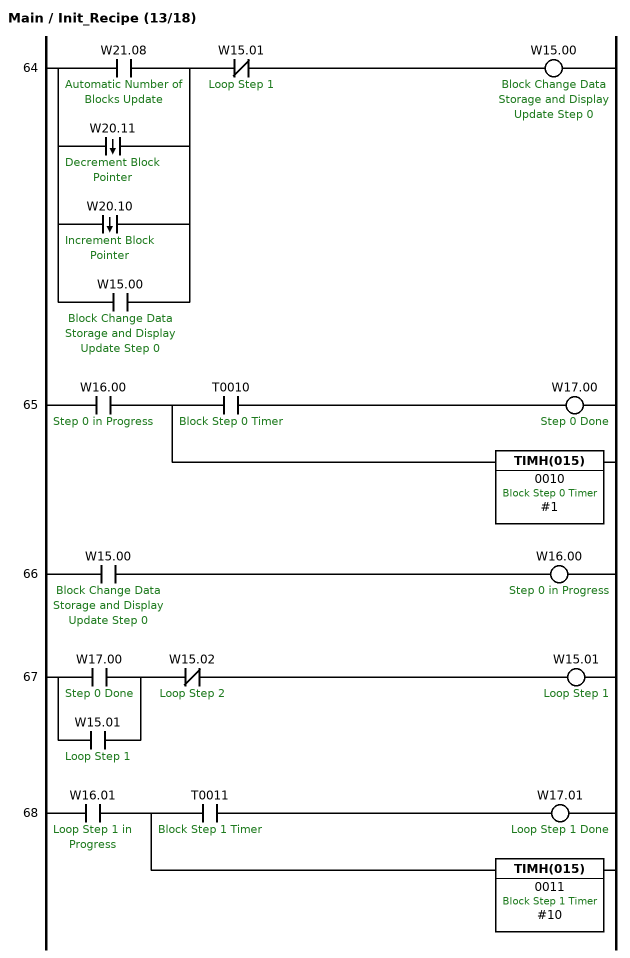
; [picture p72: Main / Init_Recipe, rungs 64-68]
; rung 64
LD W21.08  ; Automatic Number of Blocks Update
%OR W20.11  ; Decrement Block Pointer
%OR W20.10  ; Increment Block Pointer
OR W15.00  ; Block Change Data Storage and Display Update Step 0
ANDNOT W15.01  ; Loop Step 1
OUT W15.00  ; Block Change Data Storage and Display Update Step 0
; rung 65
LD W16.00  ; Step 0 in Progress
OUT TR0
AND T0010  ; Block Step 0 Timer
OUT W17.00  ; Step 0 Done
LD TR0
TIMH(015) 0010 #1  ; Block Step 0 Timer
; rung 66
LD W15.00  ; Block Change Data Storage and Display Update Step 0
OUT W16.00  ; Step 0 in Progress
; rung 67
LD W17.00  ; Step 0 Done
OR W15.01  ; Loop Step 1
ANDNOT W15.02  ; Loop Step 2
OUT W15.01  ; Loop Step 1
; rung 68
LD W16.01  ; Loop Step 1 in Progress
OUT TR0
AND T0011  ; Block Step 1 Timer
OUT W17.01  ; Loop Step 1 Done
LD TR0
TIMH(015) 0011 #10  ; Block Step 1 Timer

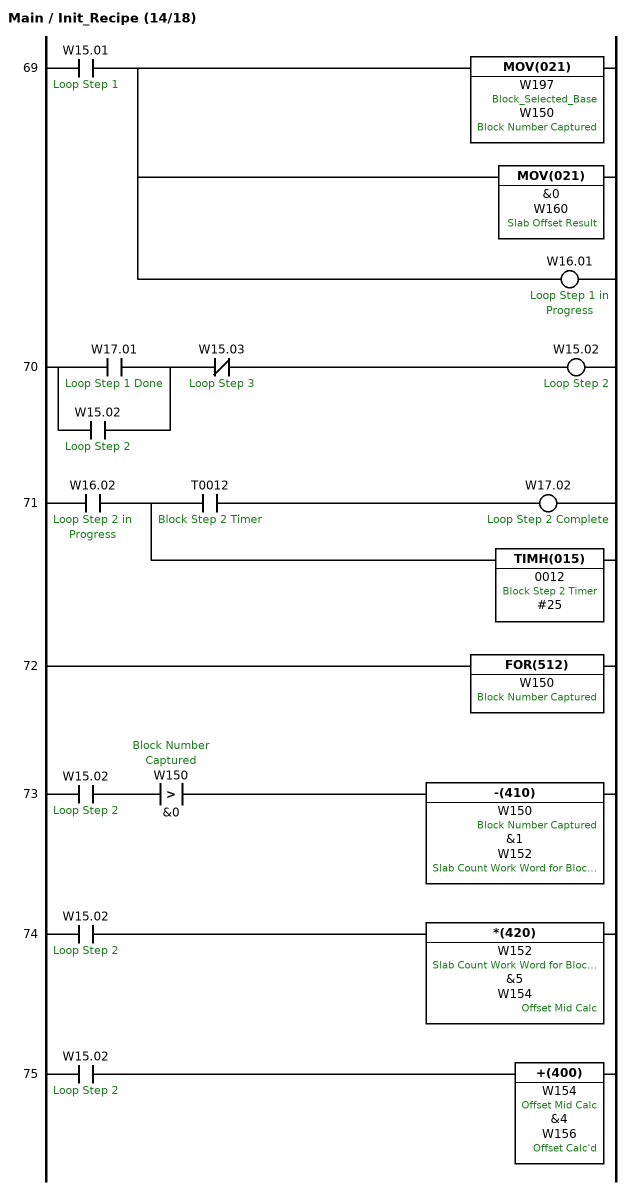
; rung 69
LD W15.01  ; Loop Step 1
MOV(021) W197 W150  ; Block_Selected_Base, Block Number Captured
MOV(021) &0 W160  ; Slab Offset Result
OUT W16.01  ; Loop Step 1 in Progress
; rung 70
LD W17.01  ; Loop Step 1 Done
OR W15.02  ; Loop Step 2
ANDNOT W15.03  ; Loop Step 3
OUT W15.02  ; Loop Step 2
; rung 71
LD W16.02  ; Loop Step 2 in Progress
OUT TR0
AND T0012  ; Block Step 2 Timer
OUT W17.02  ; Loop Step 2 Complete
LD TR0
TIMH(015) 0012 #25  ; Block Step 2 Timer
; rung 72
FOR(512) W150  ; Block Number Captured
; rung 73
LD W15.02  ; Loop Step 2
AND>(320) W150 &0  ; Block Number Captured
-(410) W150 &1 W152  ; Block Number Captured, Slab Count Work Word for Block Pointer
; rung 74
LD W15.02  ; Loop Step 2
*(420) W152 &5 W154  ; Slab Count Work Word for Block Pointer, Offset Mid Calc
; rung 75
LD W15.02  ; Loop Step 2
+(400) W154 &4 W156  ; Offset Mid Calc, Offset Calc'd

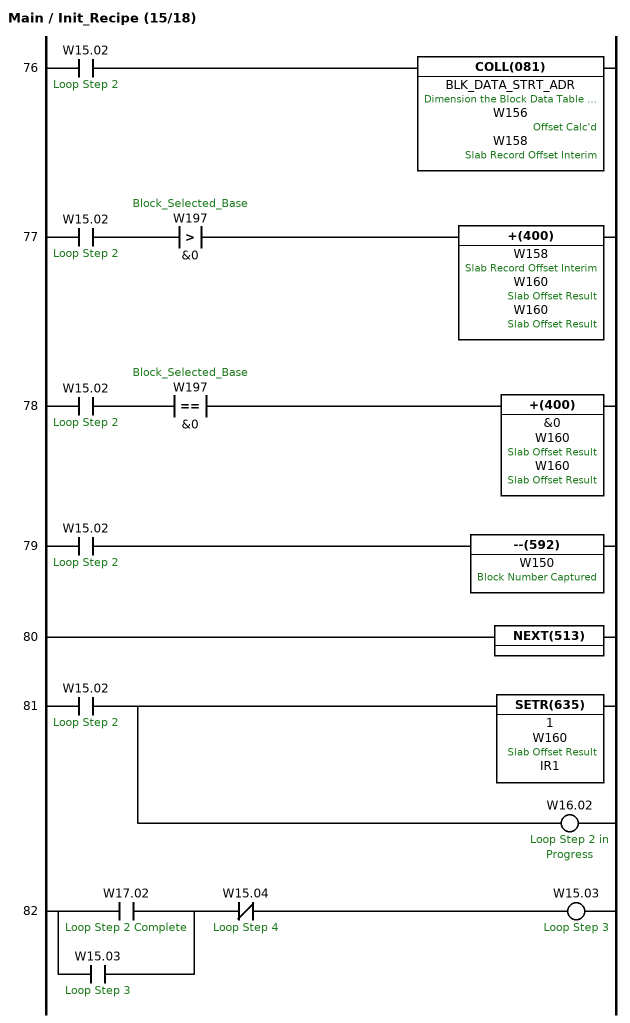
; rung 76
LD W15.02  ; Loop Step 2
COLL(081) BLK_DATA_STRT_ADR W156 W158  ; Dimension the Block Data Table - Start Address, Offset Calc'd, Slab Record Offset Interim
; rung 77
LD W15.02  ; Loop Step 2
AND>(320) W197 &0  ; Block_Selected_Base
+(400) W158 W160 W160  ; Slab Record Offset Interim, Slab Offset Result
; rung 78
LD W15.02  ; Loop Step 2
AND=(300) W197 &0  ; Block_Selected_Base
+(400) &0 W160 W160  ; Slab Offset Result
; rung 79
LD W15.02  ; Loop Step 2
--(592) W150  ; Block Number Captured
; rung 80
NEXT(513)
; rung 81
LD W15.02  ; Loop Step 2
SETR(635) 1 W160 IR1  ; Slab Offset Result
OUT W16.02  ; Loop Step 2 in Progress
; rung 82
LD W17.02  ; Loop Step 2 Complete
OR W15.03  ; Loop Step 3
ANDNOT W15.04  ; Loop Step 4
OUT W15.03  ; Loop Step 3

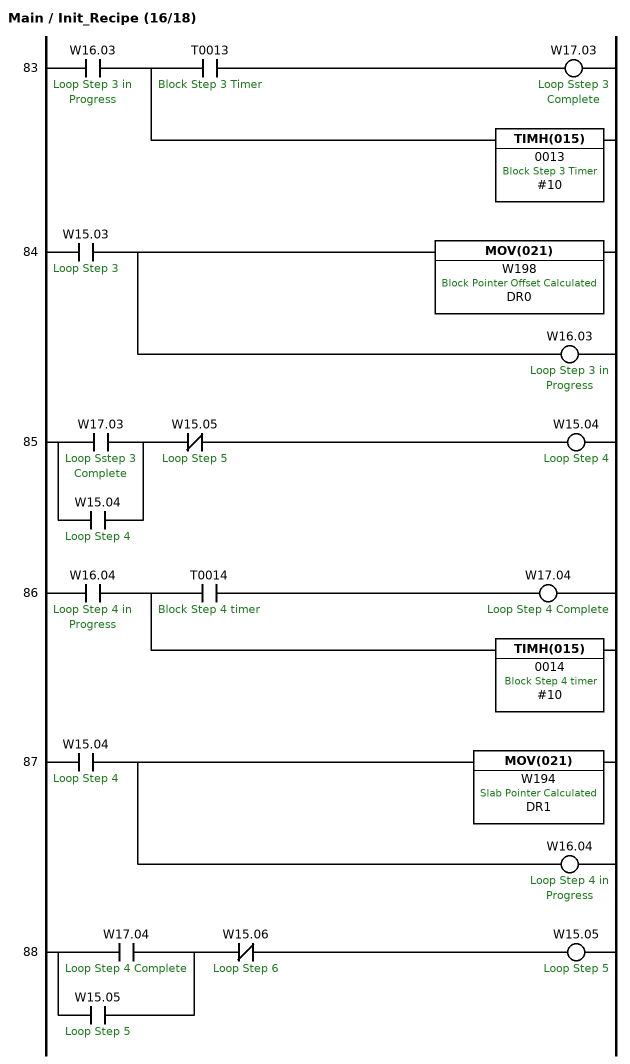
; rung 83
LD W16.03  ; Loop Step 3 in Progress
OUT TR0
AND T0013  ; Block Step 3 Timer
OUT W17.03  ; Loop Sstep 3 Complete
LD TR0
TIMH(015) 0013 #10  ; Block Step 3 Timer
; rung 84
LD W15.03  ; Loop Step 3
MOV(021) W198 DR0  ; Block Pointer Offset Calculated
OUT W16.03  ; Loop Step 3 in Progress
; rung 85
LD W17.03  ; Loop Sstep 3 Complete
OR W15.04  ; Loop Step 4
ANDNOT W15.05  ; Loop Step 5
OUT W15.04  ; Loop Step 4
; rung 86
LD W16.04  ; Loop Step 4 in Progress
OUT TR0
AND T0014  ; Block Step 4 timer
OUT W17.04  ; Loop Step 4 Complete
LD TR0
TIMH(015) 0014 #10  ; Block Step 4 timer
; rung 87
LD W15.04  ; Loop Step 4
MOV(021) W194 DR1  ; Slab Pointer Calculated
OUT W16.04  ; Loop Step 4 in Progress
; rung 88
LD W17.04  ; Loop Step 4 Complete
OR W15.05  ; Loop Step 5
ANDNOT W15.06  ; Loop Step 6
OUT W15.05  ; Loop Step 5

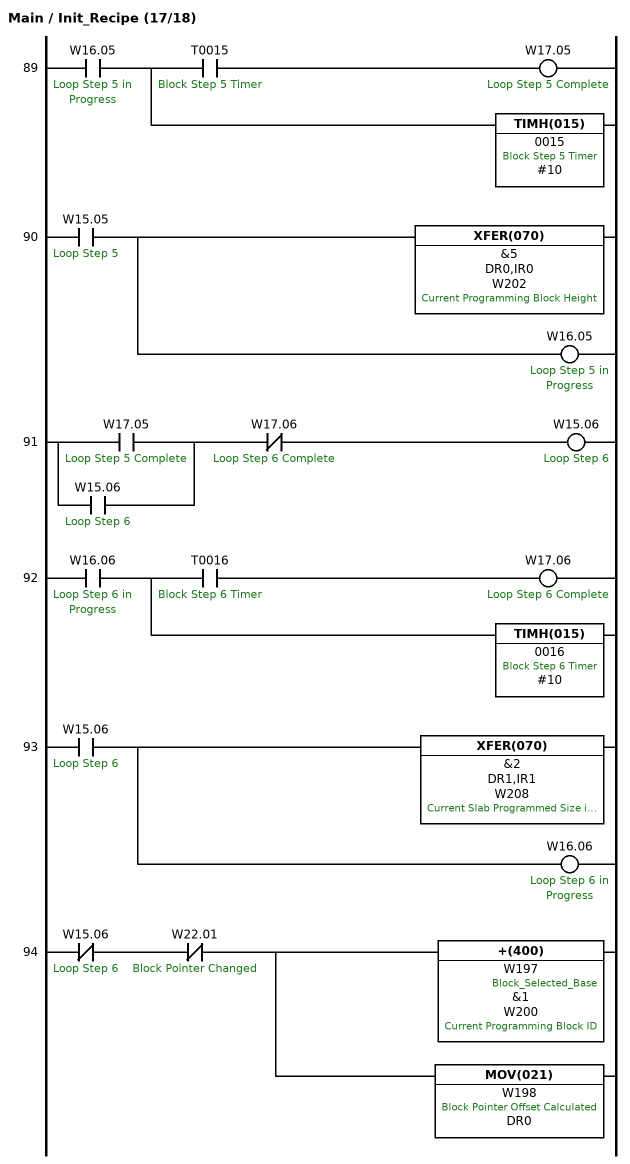
; rung 89
LD W16.05  ; Loop Step 5 in Progress
OUT TR0
AND T0015  ; Block Step 5 Timer
OUT W17.05  ; Loop Step 5 Complete
LD TR0
TIMH(015) 0015 #10  ; Block Step 5 Timer
; rung 90
LD W15.05  ; Loop Step 5
XFER(070) &5 DR0,IR0 W202  ; Current Programming Block Height
OUT W16.05  ; Loop Step 5 in Progress
; rung 91
LD W17.05  ; Loop Step 5 Complete
OR W15.06  ; Loop Step 6
ANDNOT W17.06  ; Loop Step 6 Complete
OUT W15.06  ; Loop Step 6
; rung 92
LD W16.06  ; Loop Step 6 in Progress
OUT TR0
AND T0016  ; Block Step 6 Timer
OUT W17.06  ; Loop Step 6 Complete
LD TR0
TIMH(015) 0016 #10  ; Block Step 6 Timer
; rung 93
LD W15.06  ; Loop Step 6
XFER(070) &2 DR1,IR1 W208  ; Current Slab Programmed Size in inches
OUT W16.06  ; Loop Step 6 in Progress
; rung 94
LDNOT W15.06  ; Loop Step 6
ANDNOT W22.01  ; Block Pointer Changed
+(400) W197 &1 W200  ; Block_Selected_Base, Current Programming Block ID
MOV(021) W198 DR0  ; Block Pointer Offset Calculated

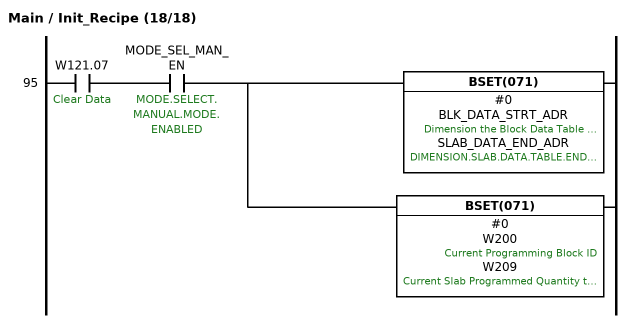
; rung 95
LD W121.07  ; Clear Data
AND MODE_SEL_MAN_EN  ; MODE.SELECT.MANUAL.MODE.ENABLED
BSET(071) #0 BLK_DATA_STRT_ADR SLAB_DATA_END_ADR  ; Dimension the Block Data Table - Start Address, DIMENSION.SLAB.DATA.TABLE.END.ADDRESS
BSET(071) #0 W200 W209  ; Current Programming Block ID, Current Slab Programmed Quantity to cut

### Section Init_Message_Display

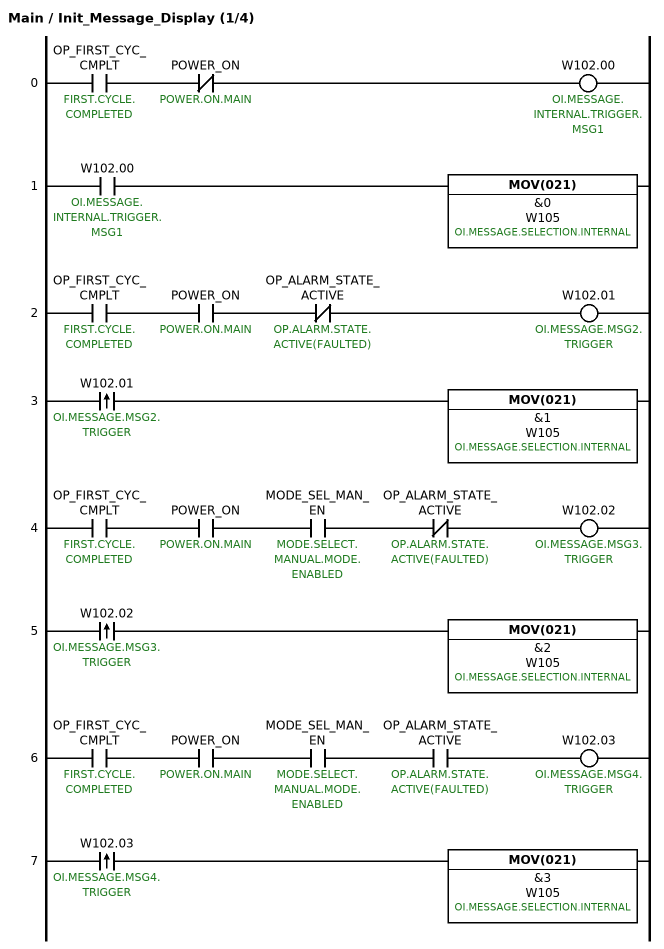
; rung 0
LD OP_FIRST_CYC_CMPLT  ; FIRST.CYCLE.COMPLETED
ANDNOT POWER_ON  ; POWER.ON.MAIN
OUT W102.00  ; OI.MESSAGE.INTERNAL.TRIGGER.MSG1
; rung 1
LD W102.00  ; OI.MESSAGE.INTERNAL.TRIGGER.MSG1
MOV(021) &0 W105  ; OI.MESSAGE.SELECTION.INTERNAL
; rung 2
LD OP_FIRST_CYC_CMPLT  ; FIRST.CYCLE.COMPLETED
AND POWER_ON  ; POWER.ON.MAIN
ANDNOT OP_ALARM_STATE_ACTIVE  ; OP.ALARM.STATE.ACTIVE(FAULTED)
OUT W102.01  ; OI.MESSAGE.MSG2.TRIGGER
; rung 3
@LD W102.01  ; OI.MESSAGE.MSG2.TRIGGER
MOV(021) &1 W105  ; OI.MESSAGE.SELECTION.INTERNAL
; rung 4
LD OP_FIRST_CYC_CMPLT  ; FIRST.CYCLE.COMPLETED
AND POWER_ON  ; POWER.ON.MAIN
AND MODE_SEL_MAN_EN  ; MODE.SELECT.MANUAL.MODE.ENABLED
ANDNOT OP_ALARM_STATE_ACTIVE  ; OP.ALARM.STATE.ACTIVE(FAULTED)
OUT W102.02  ; OI.MESSAGE.MSG3.TRIGGER
; rung 5
@LD W102.02  ; OI.MESSAGE.MSG3.TRIGGER
MOV(021) &2 W105  ; OI.MESSAGE.SELECTION.INTERNAL
; rung 6
LD OP_FIRST_CYC_CMPLT  ; FIRST.CYCLE.COMPLETED
AND POWER_ON  ; POWER.ON.MAIN
AND MODE_SEL_MAN_EN  ; MODE.SELECT.MANUAL.MODE.ENABLED
AND OP_ALARM_STATE_ACTIVE  ; OP.ALARM.STATE.ACTIVE(FAULTED)
OUT W102.03  ; OI.MESSAGE.MSG4.TRIGGER
; rung 7
@LD W102.03  ; OI.MESSAGE.MSG4.TRIGGER
MOV(021) &3 W105  ; OI.MESSAGE.SELECTION.INTERNAL

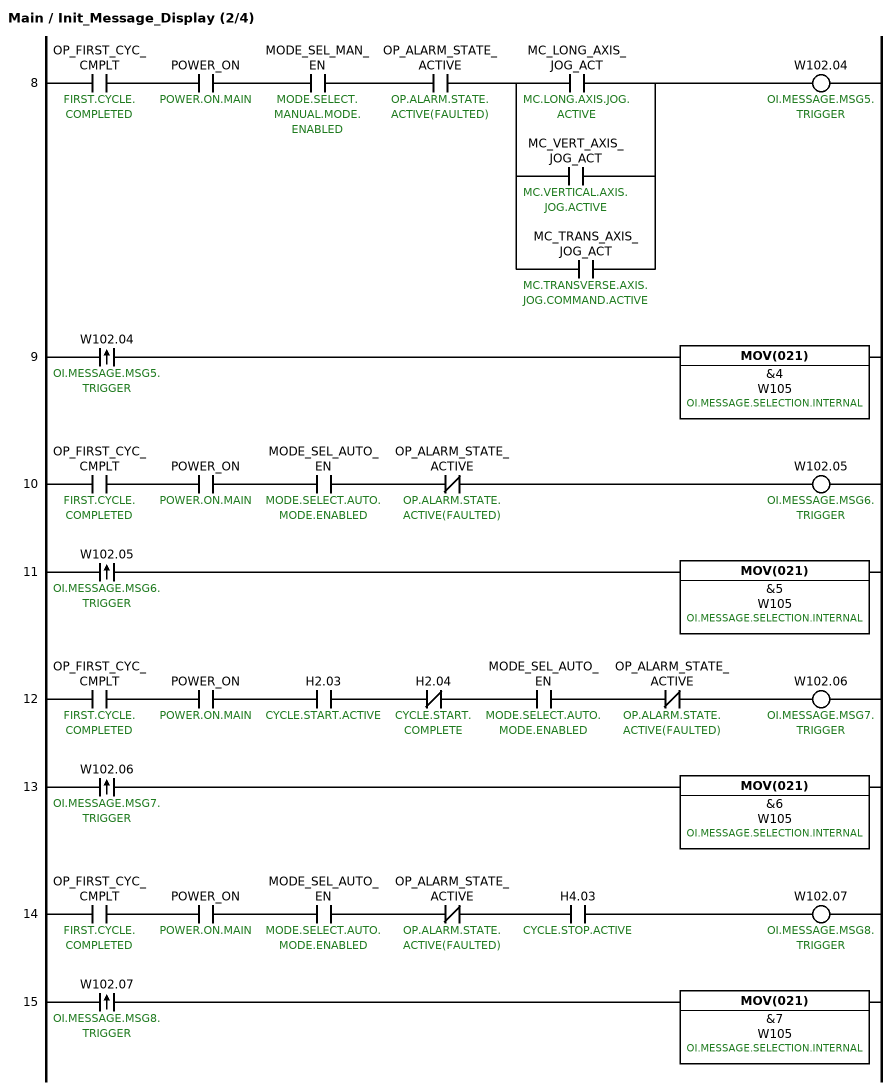
; rung 8
LD OP_FIRST_CYC_CMPLT  ; FIRST.CYCLE.COMPLETED
AND POWER_ON  ; POWER.ON.MAIN
AND MODE_SEL_MAN_EN  ; MODE.SELECT.MANUAL.MODE.ENABLED
AND OP_ALARM_STATE_ACTIVE  ; OP.ALARM.STATE.ACTIVE(FAULTED)
LD MC_LONG_AXIS_JOG_ACT  ; MC.LONG.AXIS.JOG.ACTIVE
OR MC_VERT_AXIS_JOG_ACT  ; MC.VERTICAL.AXIS.JOG.ACTIVE
OR MC_TRANS_AXIS_JOG_ACT  ; MC.TRANSVERSE.AXIS.JOG.COMMAND.ACTIVE
ANDLD
OUT W102.04  ; OI.MESSAGE.MSG5.TRIGGER
; rung 9
@LD W102.04  ; OI.MESSAGE.MSG5.TRIGGER
MOV(021) &4 W105  ; OI.MESSAGE.SELECTION.INTERNAL
; rung 10
LD OP_FIRST_CYC_CMPLT  ; FIRST.CYCLE.COMPLETED
AND POWER_ON  ; POWER.ON.MAIN
AND MODE_SEL_AUTO_EN  ; MODE.SELECT.AUTO.MODE.ENABLED
ANDNOT OP_ALARM_STATE_ACTIVE  ; OP.ALARM.STATE.ACTIVE(FAULTED)
OUT W102.05  ; OI.MESSAGE.MSG6.TRIGGER
; rung 11
@LD W102.05  ; OI.MESSAGE.MSG6.TRIGGER
MOV(021) &5 W105  ; OI.MESSAGE.SELECTION.INTERNAL
; rung 12
LD OP_FIRST_CYC_CMPLT  ; FIRST.CYCLE.COMPLETED
AND POWER_ON  ; POWER.ON.MAIN
AND H2.03  ; CYCLE.START.ACTIVE
ANDNOT H2.04  ; CYCLE.START.COMPLETE
AND MODE_SEL_AUTO_EN  ; MODE.SELECT.AUTO.MODE.ENABLED
ANDNOT OP_ALARM_STATE_ACTIVE  ; OP.ALARM.STATE.ACTIVE(FAULTED)
OUT W102.06  ; OI.MESSAGE.MSG7.TRIGGER
; rung 13
@LD W102.06  ; OI.MESSAGE.MSG7.TRIGGER
MOV(021) &6 W105  ; OI.MESSAGE.SELECTION.INTERNAL
; rung 14
LD OP_FIRST_CYC_CMPLT  ; FIRST.CYCLE.COMPLETED
AND POWER_ON  ; POWER.ON.MAIN
AND MODE_SEL_AUTO_EN  ; MODE.SELECT.AUTO.MODE.ENABLED
ANDNOT OP_ALARM_STATE_ACTIVE  ; OP.ALARM.STATE.ACTIVE(FAULTED)
AND H4.03  ; CYCLE.STOP.ACTIVE
OUT W102.07  ; OI.MESSAGE.MSG8.TRIGGER
; rung 15
@LD W102.07  ; OI.MESSAGE.MSG8.TRIGGER
MOV(021) &7 W105  ; OI.MESSAGE.SELECTION.INTERNAL

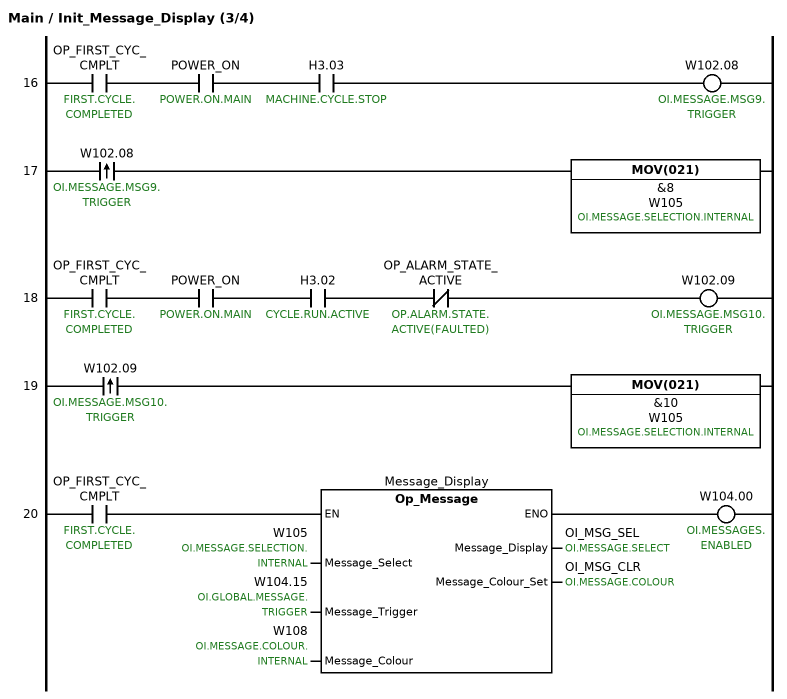
; rung 16
LD OP_FIRST_CYC_CMPLT  ; FIRST.CYCLE.COMPLETED
AND POWER_ON  ; POWER.ON.MAIN
AND H3.03  ; MACHINE.CYCLE.STOP
OUT W102.08  ; OI.MESSAGE.MSG9.TRIGGER
; rung 17
@LD W102.08  ; OI.MESSAGE.MSG9.TRIGGER
MOV(021) &8 W105  ; OI.MESSAGE.SELECTION.INTERNAL
; rung 18
LD OP_FIRST_CYC_CMPLT  ; FIRST.CYCLE.COMPLETED
AND POWER_ON  ; POWER.ON.MAIN
AND H3.02  ; CYCLE.RUN.ACTIVE
ANDNOT OP_ALARM_STATE_ACTIVE  ; OP.ALARM.STATE.ACTIVE(FAULTED)
OUT W102.09  ; OI.MESSAGE.MSG10.TRIGGER
; rung 19
@LD W102.09  ; OI.MESSAGE.MSG10.TRIGGER
MOV(021) &10 W105  ; OI.MESSAGE.SELECTION.INTERNAL
; rung 20
LD OP_FIRST_CYC_CMPLT  ; FIRST.CYCLE.COMPLETED
CALL Message_Display : Op_Message (Message_Select := W105, Message_Trigger := W104.15, Message_Colour := W108, Message_Display => OI_MSG_SEL, Message_Colour_Set => OI_MSG_CLR)  ; OI.MESSAGE.SELECTION.INTERNAL, OI.GLOBAL.MESSAGE.TRIGGER, OI.MESSAGE.COLOUR.INTERNAL, OI.MESSAGE.SELECT, OI.MESSAGE.COLOUR
OUT W104.00  ; OI.MESSAGES.ENABLED

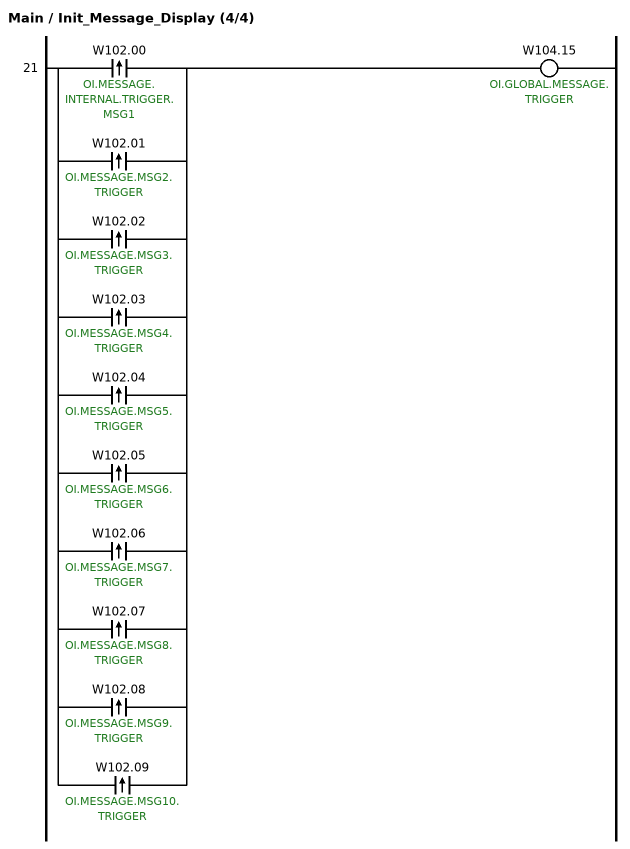
; rung 21
@LD W102.00  ; OI.MESSAGE.INTERNAL.TRIGGER.MSG1
@OR W102.01  ; OI.MESSAGE.MSG2.TRIGGER
@OR W102.02  ; OI.MESSAGE.MSG3.TRIGGER
@OR W102.03  ; OI.MESSAGE.MSG4.TRIGGER
@OR W102.04  ; OI.MESSAGE.MSG5.TRIGGER
@OR W102.05  ; OI.MESSAGE.MSG6.TRIGGER
@OR W102.06  ; OI.MESSAGE.MSG7.TRIGGER
@OR W102.07  ; OI.MESSAGE.MSG8.TRIGGER
@OR W102.08  ; OI.MESSAGE.MSG9.TRIGGER
@OR W102.09  ; OI.MESSAGE.MSG10.TRIGGER
OUT W104.15  ; OI.GLOBAL.MESSAGE.TRIGGER

### Section Init_Alarm_Display

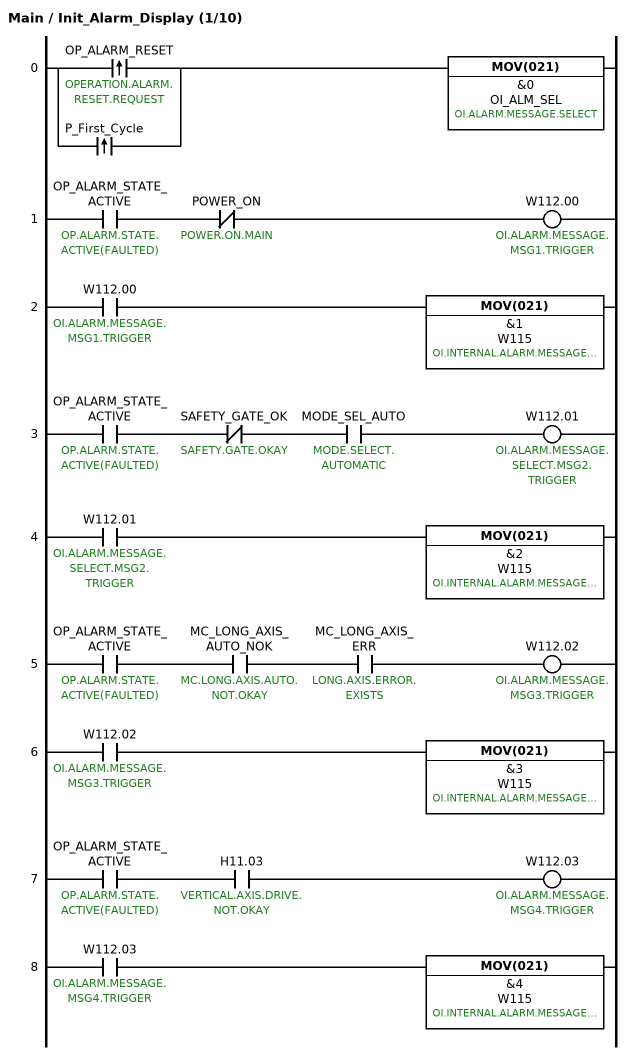
; rung 0
@LD OP_ALARM_RESET  ; OPERATION.ALARM.RESET.REQUEST
@OR P_First_Cycle
MOV(021) &0 OI_ALM_SEL  ; OI.ALARM.MESSAGE.SELECT
; rung 1
LD OP_ALARM_STATE_ACTIVE  ; OP.ALARM.STATE.ACTIVE(FAULTED)
ANDNOT POWER_ON  ; POWER.ON.MAIN
OUT W112.00  ; OI.ALARM.MESSAGE.MSG1.TRIGGER
; rung 2
LD W112.00  ; OI.ALARM.MESSAGE.MSG1.TRIGGER
MOV(021) &1 W115  ; OI.INTERNAL.ALARM.MESSAGE.SELECTION
; rung 3
LD OP_ALARM_STATE_ACTIVE  ; OP.ALARM.STATE.ACTIVE(FAULTED)
ANDNOT SAFETY_GATE_OK  ; SAFETY.GATE.OKAY
AND MODE_SEL_AUTO  ; MODE.SELECT.AUTOMATIC
OUT W112.01  ; OI.ALARM.MESSAGE.SELECT.MSG2.TRIGGER
; rung 4
LD W112.01  ; OI.ALARM.MESSAGE.SELECT.MSG2.TRIGGER
MOV(021) &2 W115  ; OI.INTERNAL.ALARM.MESSAGE.SELECTION
; rung 5
LD OP_ALARM_STATE_ACTIVE  ; OP.ALARM.STATE.ACTIVE(FAULTED)
AND MC_LONG_AXIS_AUTO_NOK  ; MC.LONG.AXIS.AUTO.NOT.OKAY
AND MC_LONG_AXIS_ERR  ; LONG.AXIS.ERROR.EXISTS
OUT W112.02  ; OI.ALARM.MESSAGE.MSG3.TRIGGER
; rung 6
LD W112.02  ; OI.ALARM.MESSAGE.MSG3.TRIGGER
MOV(021) &3 W115  ; OI.INTERNAL.ALARM.MESSAGE.SELECTION
; rung 7
LD OP_ALARM_STATE_ACTIVE  ; OP.ALARM.STATE.ACTIVE(FAULTED)
AND H11.03  ; VERTICAL.AXIS.DRIVE.NOT.OKAY
OUT W112.03  ; OI.ALARM.MESSAGE.MSG4.TRIGGER
; rung 8
LD W112.03  ; OI.ALARM.MESSAGE.MSG4.TRIGGER
MOV(021) &4 W115  ; OI.INTERNAL.ALARM.MESSAGE.SELECTION

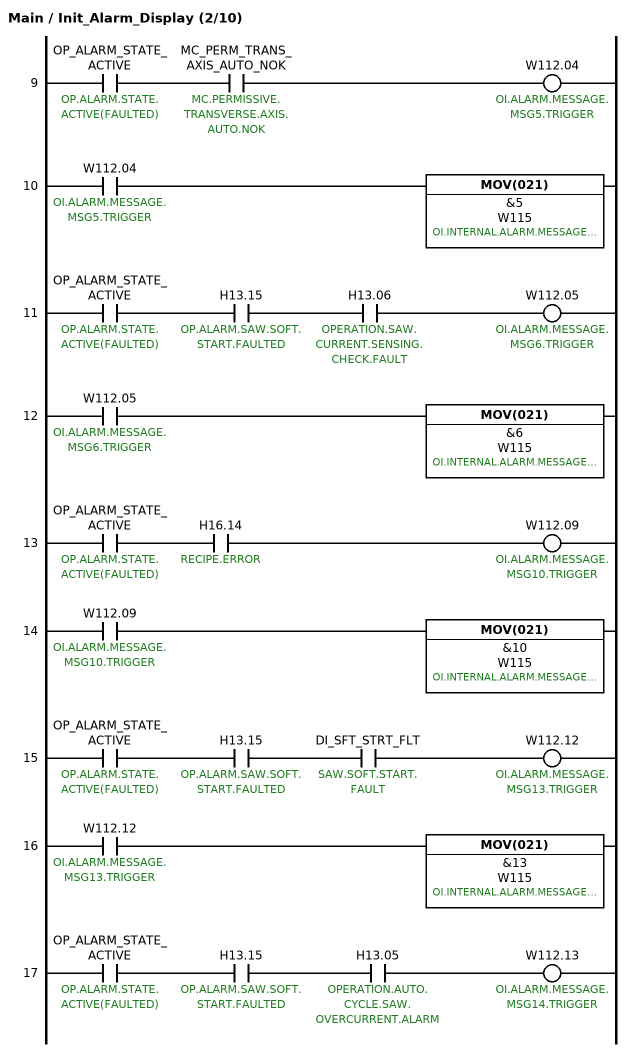
; rung 9
LD OP_ALARM_STATE_ACTIVE  ; OP.ALARM.STATE.ACTIVE(FAULTED)
AND MC_PERM_TRANS_AXIS_AUTO_NOK  ; MC.PERMISSIVE.TRANSVERSE.AXIS.AUTO.NOK
OUT W112.04  ; OI.ALARM.MESSAGE.MSG5.TRIGGER
; rung 10
LD W112.04  ; OI.ALARM.MESSAGE.MSG5.TRIGGER
MOV(021) &5 W115  ; OI.INTERNAL.ALARM.MESSAGE.SELECTION
; rung 11
LD OP_ALARM_STATE_ACTIVE  ; OP.ALARM.STATE.ACTIVE(FAULTED)
AND H13.15  ; OP.ALARM.SAW.SOFT.START.FAULTED
AND H13.06  ; OPERATION.SAW.CURRENT.SENSING.CHECK.FAULT
OUT W112.05  ; OI.ALARM.MESSAGE.MSG6.TRIGGER
; rung 12
LD W112.05  ; OI.ALARM.MESSAGE.MSG6.TRIGGER
MOV(021) &6 W115  ; OI.INTERNAL.ALARM.MESSAGE.SELECTION
; rung 13
LD OP_ALARM_STATE_ACTIVE  ; OP.ALARM.STATE.ACTIVE(FAULTED)
AND H16.14  ; RECIPE.ERROR
OUT W112.09  ; OI.ALARM.MESSAGE.MSG10.TRIGGER
; rung 14
LD W112.09  ; OI.ALARM.MESSAGE.MSG10.TRIGGER
MOV(021) &10 W115  ; OI.INTERNAL.ALARM.MESSAGE.SELECTION
; rung 15
LD OP_ALARM_STATE_ACTIVE  ; OP.ALARM.STATE.ACTIVE(FAULTED)
AND H13.15  ; OP.ALARM.SAW.SOFT.START.FAULTED
AND DI_SFT_STRT_FLT  ; SAW.SOFT.START.FAULT
OUT W112.12  ; OI.ALARM.MESSAGE.MSG13.TRIGGER
; rung 16
LD W112.12  ; OI.ALARM.MESSAGE.MSG13.TRIGGER
MOV(021) &13 W115  ; OI.INTERNAL.ALARM.MESSAGE.SELECTION
; rung 17
LD OP_ALARM_STATE_ACTIVE  ; OP.ALARM.STATE.ACTIVE(FAULTED)
AND H13.15  ; OP.ALARM.SAW.SOFT.START.FAULTED
AND H13.05  ; OPERATION.AUTO.CYCLE.SAW.OVERCURRENT.ALARM
OUT W112.13  ; OI.ALARM.MESSAGE.MSG14.TRIGGER

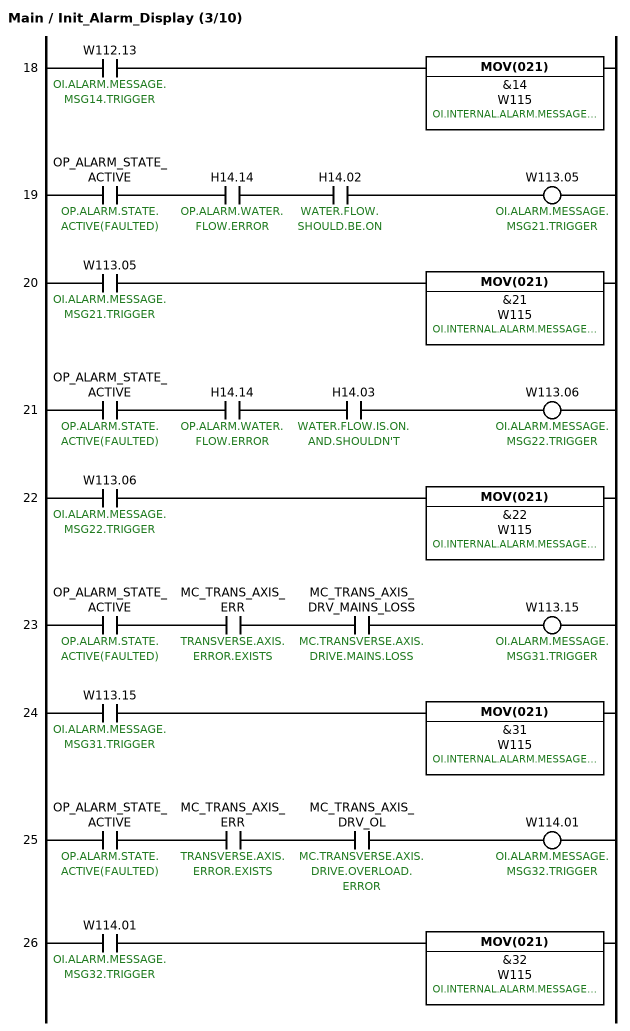
; rung 18
LD W112.13  ; OI.ALARM.MESSAGE.MSG14.TRIGGER
MOV(021) &14 W115  ; OI.INTERNAL.ALARM.MESSAGE.SELECTION
; rung 19
LD OP_ALARM_STATE_ACTIVE  ; OP.ALARM.STATE.ACTIVE(FAULTED)
AND H14.14  ; OP.ALARM.WATER.FLOW.ERROR
AND H14.02  ; WATER.FLOW.SHOULD.BE.ON
OUT W113.05  ; OI.ALARM.MESSAGE.MSG21.TRIGGER
; rung 20
LD W113.05  ; OI.ALARM.MESSAGE.MSG21.TRIGGER
MOV(021) &21 W115  ; OI.INTERNAL.ALARM.MESSAGE.SELECTION
; rung 21
LD OP_ALARM_STATE_ACTIVE  ; OP.ALARM.STATE.ACTIVE(FAULTED)
AND H14.14  ; OP.ALARM.WATER.FLOW.ERROR
AND H14.03  ; WATER.FLOW.IS.ON.AND.SHOULDN'T
OUT W113.06  ; OI.ALARM.MESSAGE.MSG22.TRIGGER
; rung 22
LD W113.06  ; OI.ALARM.MESSAGE.MSG22.TRIGGER
MOV(021) &22 W115  ; OI.INTERNAL.ALARM.MESSAGE.SELECTION
; rung 23
LD OP_ALARM_STATE_ACTIVE  ; OP.ALARM.STATE.ACTIVE(FAULTED)
AND MC_TRANS_AXIS_ERR  ; TRANSVERSE.AXIS.ERROR.EXISTS
AND MC_TRANS_AXIS_DRV_MAINS_LOSS  ; MC.TRANSVERSE.AXIS.DRIVE.MAINS.LOSS
OUT W113.15  ; OI.ALARM.MESSAGE.MSG31.TRIGGER
; rung 24
LD W113.15  ; OI.ALARM.MESSAGE.MSG31.TRIGGER
MOV(021) &31 W115  ; OI.INTERNAL.ALARM.MESSAGE.SELECTION
; rung 25
LD OP_ALARM_STATE_ACTIVE  ; OP.ALARM.STATE.ACTIVE(FAULTED)
AND MC_TRANS_AXIS_ERR  ; TRANSVERSE.AXIS.ERROR.EXISTS
AND MC_TRANS_AXIS_DRV_OL  ; MC.TRANSVERSE.AXIS.DRIVE.OVERLOAD.ERROR
OUT W114.01  ; OI.ALARM.MESSAGE.MSG32.TRIGGER
; rung 26
LD W114.01  ; OI.ALARM.MESSAGE.MSG32.TRIGGER
MOV(021) &32 W115  ; OI.INTERNAL.ALARM.MESSAGE.SELECTION

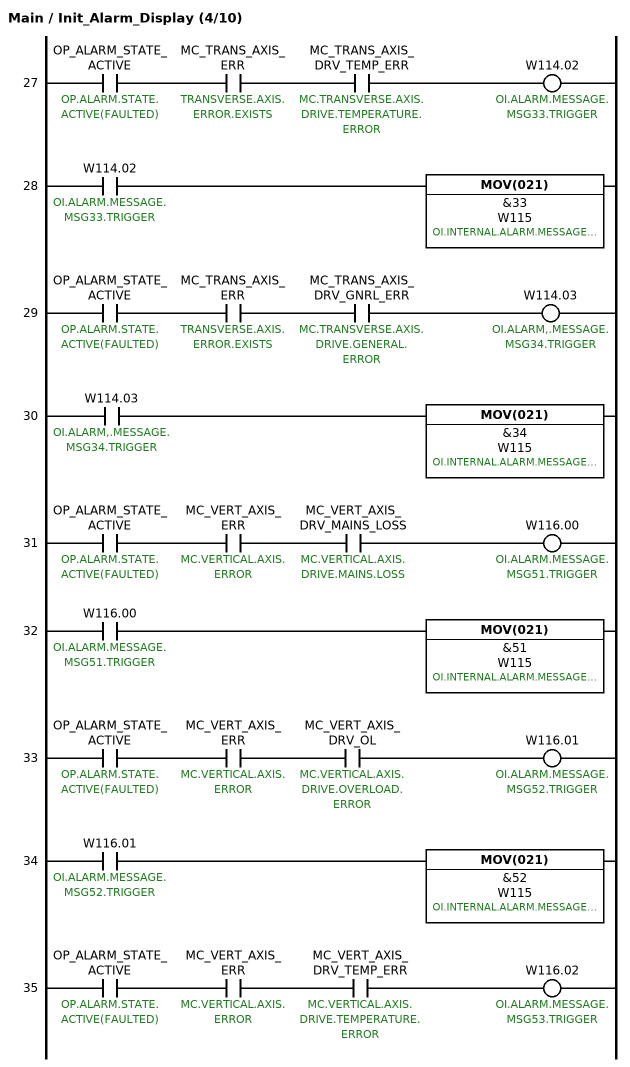
; rung 27
LD OP_ALARM_STATE_ACTIVE  ; OP.ALARM.STATE.ACTIVE(FAULTED)
AND MC_TRANS_AXIS_ERR  ; TRANSVERSE.AXIS.ERROR.EXISTS
AND MC_TRANS_AXIS_DRV_TEMP_ERR  ; MC.TRANSVERSE.AXIS.DRIVE.TEMPERATURE.ERROR
OUT W114.02  ; OI.ALARM.MESSAGE.MSG33.TRIGGER
; rung 28
LD W114.02  ; OI.ALARM.MESSAGE.MSG33.TRIGGER
MOV(021) &33 W115  ; OI.INTERNAL.ALARM.MESSAGE.SELECTION
; rung 29
LD OP_ALARM_STATE_ACTIVE  ; OP.ALARM.STATE.ACTIVE(FAULTED)
AND MC_TRANS_AXIS_ERR  ; TRANSVERSE.AXIS.ERROR.EXISTS
AND MC_TRANS_AXIS_DRV_GNRL_ERR  ; MC.TRANSVERSE.AXIS.DRIVE.GENERAL.ERROR
OUT W114.03  ; OI.ALARM,.MESSAGE.MSG34.TRIGGER
; rung 30
LD W114.03  ; OI.ALARM,.MESSAGE.MSG34.TRIGGER
MOV(021) &34 W115  ; OI.INTERNAL.ALARM.MESSAGE.SELECTION
; rung 31
LD OP_ALARM_STATE_ACTIVE  ; OP.ALARM.STATE.ACTIVE(FAULTED)
AND MC_VERT_AXIS_ERR  ; MC.VERTICAL.AXIS.ERROR
AND MC_VERT_AXIS_DRV_MAINS_LOSS  ; MC.VERTICAL.AXIS.DRIVE.MAINS.LOSS
OUT W116.00  ; OI.ALARM.MESSAGE.MSG51.TRIGGER
; rung 32
LD W116.00  ; OI.ALARM.MESSAGE.MSG51.TRIGGER
MOV(021) &51 W115  ; OI.INTERNAL.ALARM.MESSAGE.SELECTION
; rung 33
LD OP_ALARM_STATE_ACTIVE  ; OP.ALARM.STATE.ACTIVE(FAULTED)
AND MC_VERT_AXIS_ERR  ; MC.VERTICAL.AXIS.ERROR
AND MC_VERT_AXIS_DRV_OL  ; MC.VERTICAL.AXIS.DRIVE.OVERLOAD.ERROR
OUT W116.01  ; OI.ALARM.MESSAGE.MSG52.TRIGGER
; rung 34
LD W116.01  ; OI.ALARM.MESSAGE.MSG52.TRIGGER
MOV(021) &52 W115  ; OI.INTERNAL.ALARM.MESSAGE.SELECTION
; rung 35
LD OP_ALARM_STATE_ACTIVE  ; OP.ALARM.STATE.ACTIVE(FAULTED)
AND MC_VERT_AXIS_ERR  ; MC.VERTICAL.AXIS.ERROR
AND MC_VERT_AXIS_DRV_TEMP_ERR  ; MC.VERTICAL.AXIS.DRIVE.TEMPERATURE.ERROR
OUT W116.02  ; OI.ALARM.MESSAGE.MSG53.TRIGGER

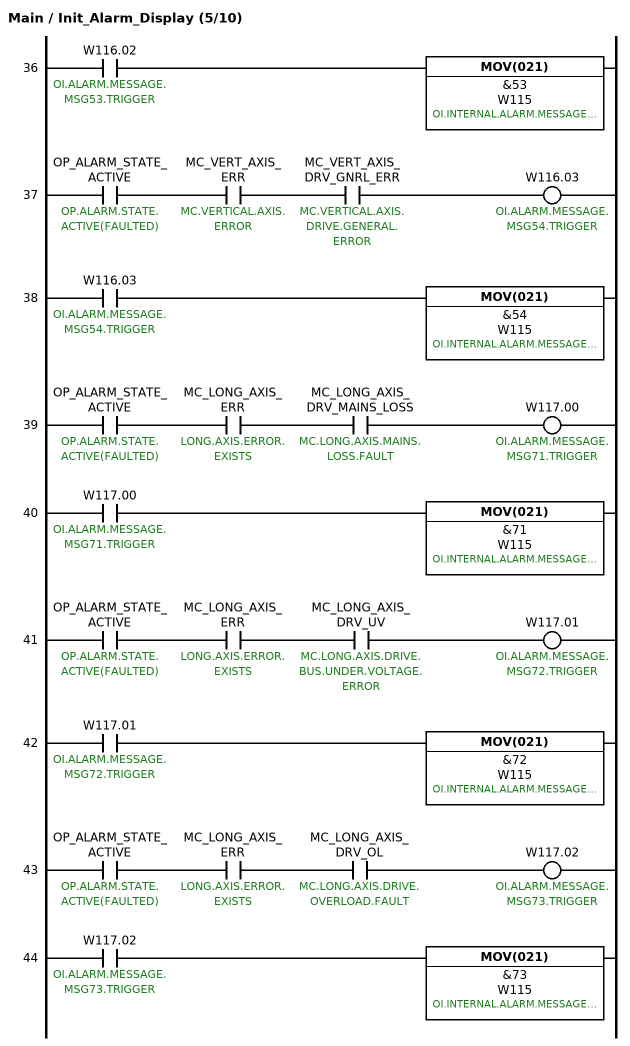
; rung 36
LD W116.02  ; OI.ALARM.MESSAGE.MSG53.TRIGGER
MOV(021) &53 W115  ; OI.INTERNAL.ALARM.MESSAGE.SELECTION
; rung 37
LD OP_ALARM_STATE_ACTIVE  ; OP.ALARM.STATE.ACTIVE(FAULTED)
AND MC_VERT_AXIS_ERR  ; MC.VERTICAL.AXIS.ERROR
AND MC_VERT_AXIS_DRV_GNRL_ERR  ; MC.VERTICAL.AXIS.DRIVE.GENERAL.ERROR
OUT W116.03  ; OI.ALARM.MESSAGE.MSG54.TRIGGER
; rung 38
LD W116.03  ; OI.ALARM.MESSAGE.MSG54.TRIGGER
MOV(021) &54 W115  ; OI.INTERNAL.ALARM.MESSAGE.SELECTION
; rung 39
LD OP_ALARM_STATE_ACTIVE  ; OP.ALARM.STATE.ACTIVE(FAULTED)
AND MC_LONG_AXIS_ERR  ; LONG.AXIS.ERROR.EXISTS
AND MC_LONG_AXIS_DRV_MAINS_LOSS  ; MC.LONG.AXIS.MAINS.LOSS.FAULT
OUT W117.00  ; OI.ALARM.MESSAGE.MSG71.TRIGGER
; rung 40
LD W117.00  ; OI.ALARM.MESSAGE.MSG71.TRIGGER
MOV(021) &71 W115  ; OI.INTERNAL.ALARM.MESSAGE.SELECTION
; rung 41
LD OP_ALARM_STATE_ACTIVE  ; OP.ALARM.STATE.ACTIVE(FAULTED)
AND MC_LONG_AXIS_ERR  ; LONG.AXIS.ERROR.EXISTS
AND MC_LONG_AXIS_DRV_UV  ; MC.LONG.AXIS.DRIVE.BUS.UNDER.VOLTAGE.ERROR
OUT W117.01  ; OI.ALARM.MESSAGE.MSG72.TRIGGER
; rung 42
LD W117.01  ; OI.ALARM.MESSAGE.MSG72.TRIGGER
MOV(021) &72 W115  ; OI.INTERNAL.ALARM.MESSAGE.SELECTION
; rung 43
LD OP_ALARM_STATE_ACTIVE  ; OP.ALARM.STATE.ACTIVE(FAULTED)
AND MC_LONG_AXIS_ERR  ; LONG.AXIS.ERROR.EXISTS
AND MC_LONG_AXIS_DRV_OL  ; MC.LONG.AXIS.DRIVE.OVERLOAD.FAULT
OUT W117.02  ; OI.ALARM.MESSAGE.MSG73.TRIGGER
; rung 44
LD W117.02  ; OI.ALARM.MESSAGE.MSG73.TRIGGER
MOV(021) &73 W115  ; OI.INTERNAL.ALARM.MESSAGE.SELECTION

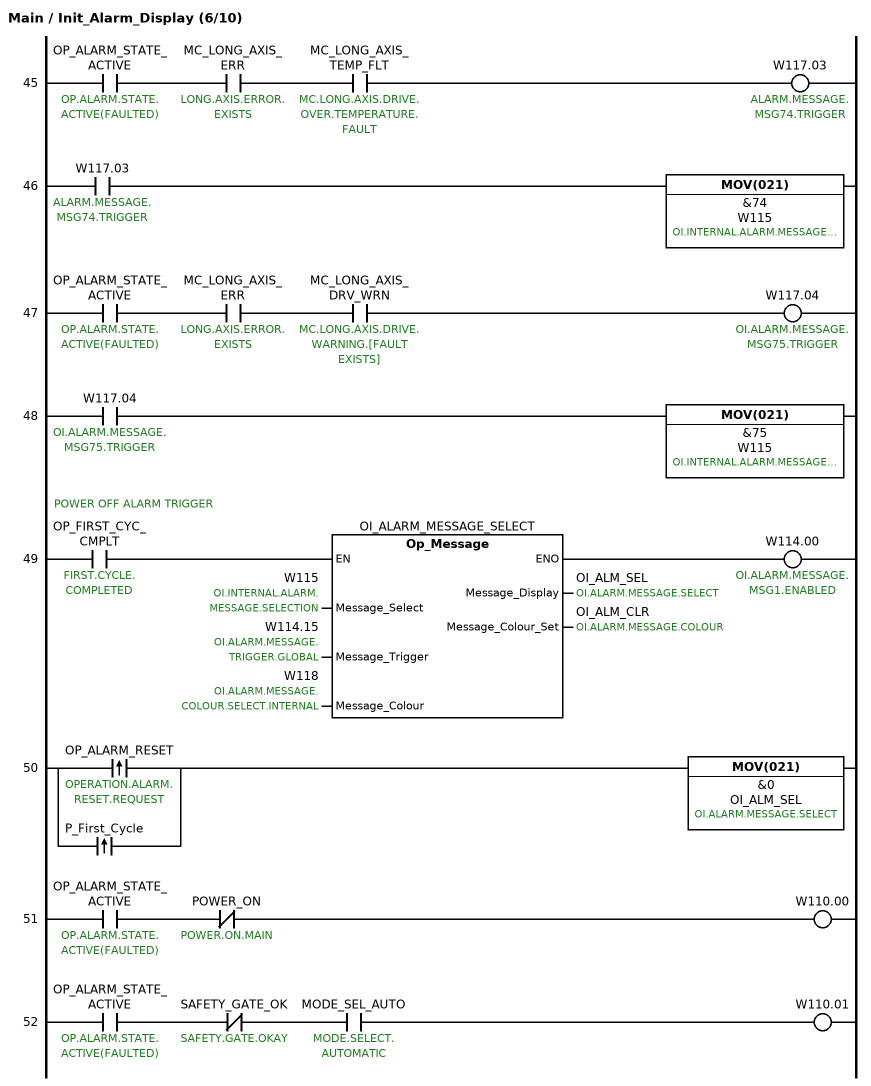
; rung 45
LD OP_ALARM_STATE_ACTIVE  ; OP.ALARM.STATE.ACTIVE(FAULTED)
AND MC_LONG_AXIS_ERR  ; LONG.AXIS.ERROR.EXISTS
AND MC_LONG_AXIS_TEMP_FLT  ; MC.LONG.AXIS.DRIVE.OVER.TEMPERATURE.FAULT
OUT W117.03  ; ALARM.MESSAGE.MSG74.TRIGGER
; rung 46
LD W117.03  ; ALARM.MESSAGE.MSG74.TRIGGER
MOV(021) &74 W115  ; OI.INTERNAL.ALARM.MESSAGE.SELECTION
; rung 47
LD OP_ALARM_STATE_ACTIVE  ; OP.ALARM.STATE.ACTIVE(FAULTED)
AND MC_LONG_AXIS_ERR  ; LONG.AXIS.ERROR.EXISTS
AND MC_LONG_AXIS_DRV_WRN  ; MC.LONG.AXIS.DRIVE.WARNING.[FAULT EXISTS]
OUT W117.04  ; OI.ALARM.MESSAGE.MSG75.TRIGGER
; rung 48
LD W117.04  ; OI.ALARM.MESSAGE.MSG75.TRIGGER
MOV(021) &75 W115  ; OI.INTERNAL.ALARM.MESSAGE.SELECTION
; rung 49: POWER OFF ALARM TRIGGER
LD OP_FIRST_CYC_CMPLT  ; FIRST.CYCLE.COMPLETED
CALL OI_ALARM_MESSAGE_SELECT : Op_Message (Message_Select := W115, Message_Trigger := W114.15, Message_Colour := W118, Message_Display => OI_ALM_SEL, Message_Colour_Set => OI_ALM_CLR)  ; OI.INTERNAL.ALARM.MESSAGE.SELECTION, OI.ALARM.MESSAGE.TRIGGER.GLOBAL, OI.ALARM.MESSAGE.COLOUR.SELECT.INTERNAL, OI.ALARM.MESSAGE.SELECT, OI.ALARM.MESSAGE.COLOUR
OUT W114.00  ; OI.ALARM.MESSAGE.MSG1.ENABLED
; rung 50
@LD OP_ALARM_RESET  ; OPERATION.ALARM.RESET.REQUEST
@OR P_First_Cycle
MOV(021) &0 OI_ALM_SEL  ; OI.ALARM.MESSAGE.SELECT
; rung 51
LD OP_ALARM_STATE_ACTIVE  ; OP.ALARM.STATE.ACTIVE(FAULTED)
ANDNOT POWER_ON  ; POWER.ON.MAIN
OUT W110.00
; rung 52
LD OP_ALARM_STATE_ACTIVE  ; OP.ALARM.STATE.ACTIVE(FAULTED)
ANDNOT SAFETY_GATE_OK  ; SAFETY.GATE.OKAY
AND MODE_SEL_AUTO  ; MODE.SELECT.AUTOMATIC
OUT W110.01

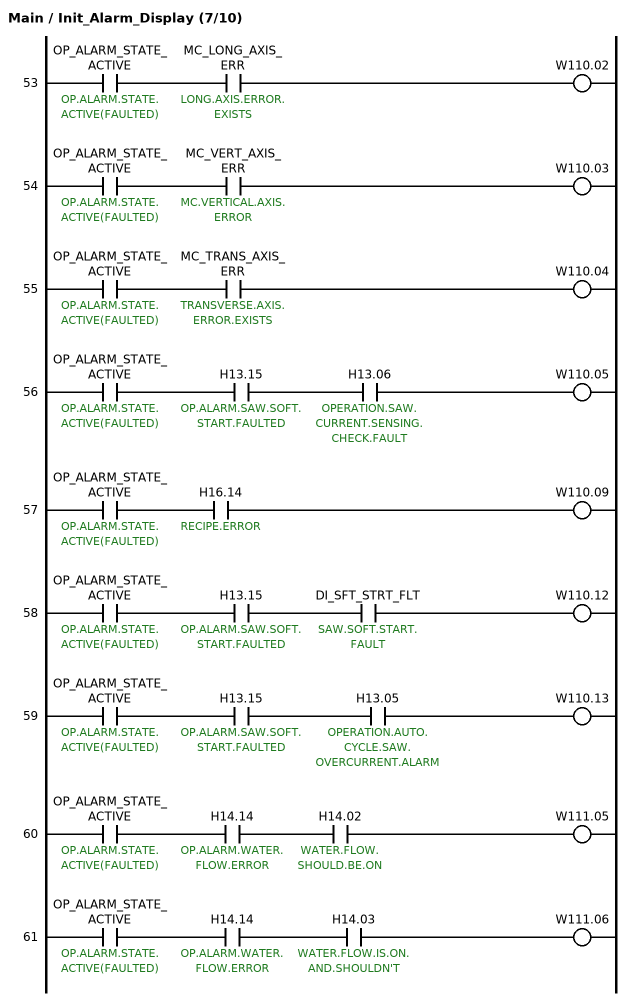
; rung 53
LD OP_ALARM_STATE_ACTIVE  ; OP.ALARM.STATE.ACTIVE(FAULTED)
AND MC_LONG_AXIS_ERR  ; LONG.AXIS.ERROR.EXISTS
OUT W110.02
; rung 54
LD OP_ALARM_STATE_ACTIVE  ; OP.ALARM.STATE.ACTIVE(FAULTED)
AND MC_VERT_AXIS_ERR  ; MC.VERTICAL.AXIS.ERROR
OUT W110.03
; rung 55
LD OP_ALARM_STATE_ACTIVE  ; OP.ALARM.STATE.ACTIVE(FAULTED)
AND MC_TRANS_AXIS_ERR  ; TRANSVERSE.AXIS.ERROR.EXISTS
OUT W110.04
; rung 56
LD OP_ALARM_STATE_ACTIVE  ; OP.ALARM.STATE.ACTIVE(FAULTED)
AND H13.15  ; OP.ALARM.SAW.SOFT.START.FAULTED
AND H13.06  ; OPERATION.SAW.CURRENT.SENSING.CHECK.FAULT
OUT W110.05
; rung 57
LD OP_ALARM_STATE_ACTIVE  ; OP.ALARM.STATE.ACTIVE(FAULTED)
AND H16.14  ; RECIPE.ERROR
OUT W110.09
; rung 58
LD OP_ALARM_STATE_ACTIVE  ; OP.ALARM.STATE.ACTIVE(FAULTED)
AND H13.15  ; OP.ALARM.SAW.SOFT.START.FAULTED
AND DI_SFT_STRT_FLT  ; SAW.SOFT.START.FAULT
OUT W110.12
; rung 59
LD OP_ALARM_STATE_ACTIVE  ; OP.ALARM.STATE.ACTIVE(FAULTED)
AND H13.15  ; OP.ALARM.SAW.SOFT.START.FAULTED
AND H13.05  ; OPERATION.AUTO.CYCLE.SAW.OVERCURRENT.ALARM
OUT W110.13
; rung 60
LD OP_ALARM_STATE_ACTIVE  ; OP.ALARM.STATE.ACTIVE(FAULTED)
AND H14.14  ; OP.ALARM.WATER.FLOW.ERROR
AND H14.02  ; WATER.FLOW.SHOULD.BE.ON
OUT W111.05
; rung 61
LD OP_ALARM_STATE_ACTIVE  ; OP.ALARM.STATE.ACTIVE(FAULTED)
AND H14.14  ; OP.ALARM.WATER.FLOW.ERROR
AND H14.03  ; WATER.FLOW.IS.ON.AND.SHOULDN'T
OUT W111.06

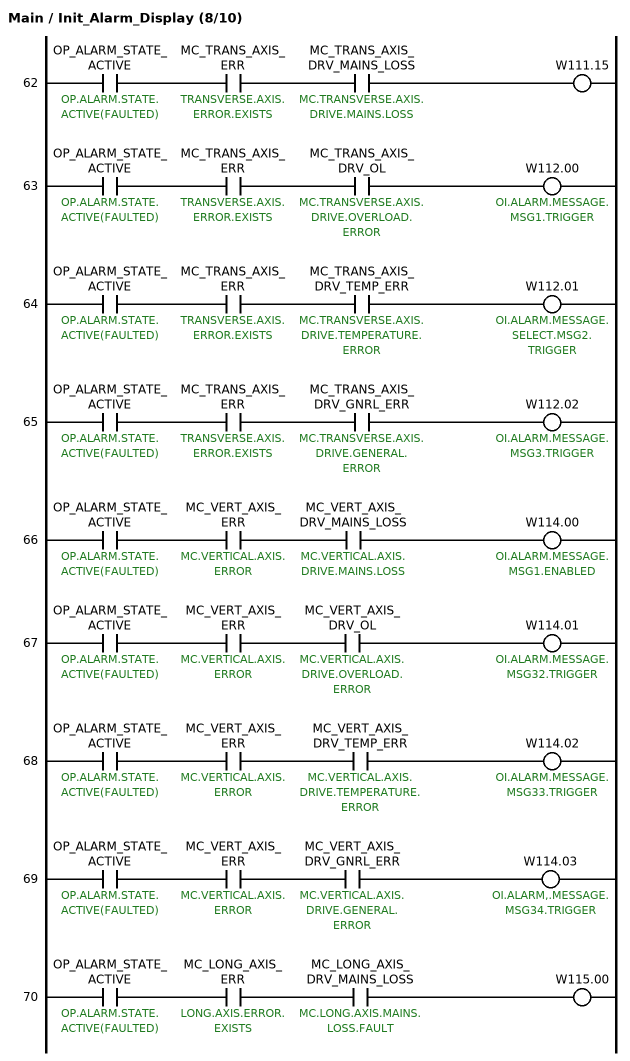
; rung 62
LD OP_ALARM_STATE_ACTIVE  ; OP.ALARM.STATE.ACTIVE(FAULTED)
AND MC_TRANS_AXIS_ERR  ; TRANSVERSE.AXIS.ERROR.EXISTS
AND MC_TRANS_AXIS_DRV_MAINS_LOSS  ; MC.TRANSVERSE.AXIS.DRIVE.MAINS.LOSS
OUT W111.15
; rung 63
LD OP_ALARM_STATE_ACTIVE  ; OP.ALARM.STATE.ACTIVE(FAULTED)
AND MC_TRANS_AXIS_ERR  ; TRANSVERSE.AXIS.ERROR.EXISTS
AND MC_TRANS_AXIS_DRV_OL  ; MC.TRANSVERSE.AXIS.DRIVE.OVERLOAD.ERROR
OUT W112.00  ; OI.ALARM.MESSAGE.MSG1.TRIGGER
; rung 64
LD OP_ALARM_STATE_ACTIVE  ; OP.ALARM.STATE.ACTIVE(FAULTED)
AND MC_TRANS_AXIS_ERR  ; TRANSVERSE.AXIS.ERROR.EXISTS
AND MC_TRANS_AXIS_DRV_TEMP_ERR  ; MC.TRANSVERSE.AXIS.DRIVE.TEMPERATURE.ERROR
OUT W112.01  ; OI.ALARM.MESSAGE.SELECT.MSG2.TRIGGER
; rung 65
LD OP_ALARM_STATE_ACTIVE  ; OP.ALARM.STATE.ACTIVE(FAULTED)
AND MC_TRANS_AXIS_ERR  ; TRANSVERSE.AXIS.ERROR.EXISTS
AND MC_TRANS_AXIS_DRV_GNRL_ERR  ; MC.TRANSVERSE.AXIS.DRIVE.GENERAL.ERROR
OUT W112.02  ; OI.ALARM.MESSAGE.MSG3.TRIGGER
; rung 66
LD OP_ALARM_STATE_ACTIVE  ; OP.ALARM.STATE.ACTIVE(FAULTED)
AND MC_VERT_AXIS_ERR  ; MC.VERTICAL.AXIS.ERROR
AND MC_VERT_AXIS_DRV_MAINS_LOSS  ; MC.VERTICAL.AXIS.DRIVE.MAINS.LOSS
OUT W114.00  ; OI.ALARM.MESSAGE.MSG1.ENABLED
; rung 67
LD OP_ALARM_STATE_ACTIVE  ; OP.ALARM.STATE.ACTIVE(FAULTED)
AND MC_VERT_AXIS_ERR  ; MC.VERTICAL.AXIS.ERROR
AND MC_VERT_AXIS_DRV_OL  ; MC.VERTICAL.AXIS.DRIVE.OVERLOAD.ERROR
OUT W114.01  ; OI.ALARM.MESSAGE.MSG32.TRIGGER
; rung 68
LD OP_ALARM_STATE_ACTIVE  ; OP.ALARM.STATE.ACTIVE(FAULTED)
AND MC_VERT_AXIS_ERR  ; MC.VERTICAL.AXIS.ERROR
AND MC_VERT_AXIS_DRV_TEMP_ERR  ; MC.VERTICAL.AXIS.DRIVE.TEMPERATURE.ERROR
OUT W114.02  ; OI.ALARM.MESSAGE.MSG33.TRIGGER
; rung 69
LD OP_ALARM_STATE_ACTIVE  ; OP.ALARM.STATE.ACTIVE(FAULTED)
AND MC_VERT_AXIS_ERR  ; MC.VERTICAL.AXIS.ERROR
AND MC_VERT_AXIS_DRV_GNRL_ERR  ; MC.VERTICAL.AXIS.DRIVE.GENERAL.ERROR
OUT W114.03  ; OI.ALARM,.MESSAGE.MSG34.TRIGGER
; rung 70
LD OP_ALARM_STATE_ACTIVE  ; OP.ALARM.STATE.ACTIVE(FAULTED)
AND MC_LONG_AXIS_ERR  ; LONG.AXIS.ERROR.EXISTS
AND MC_LONG_AXIS_DRV_MAINS_LOSS  ; MC.LONG.AXIS.MAINS.LOSS.FAULT
OUT W115.00

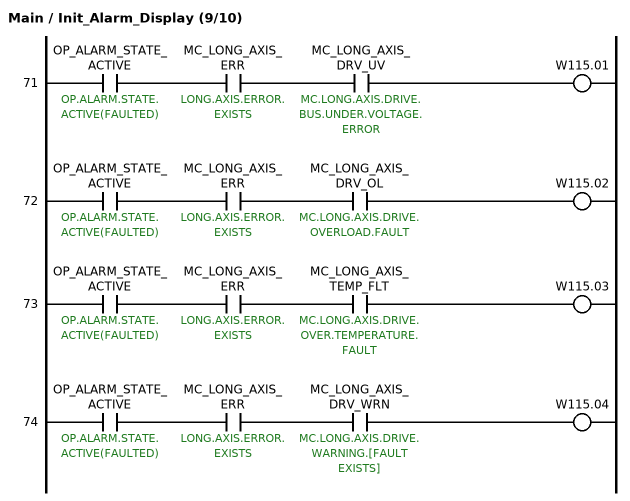
; rung 71
LD OP_ALARM_STATE_ACTIVE  ; OP.ALARM.STATE.ACTIVE(FAULTED)
AND MC_LONG_AXIS_ERR  ; LONG.AXIS.ERROR.EXISTS
AND MC_LONG_AXIS_DRV_UV  ; MC.LONG.AXIS.DRIVE.BUS.UNDER.VOLTAGE.ERROR
OUT W115.01
; rung 72
LD OP_ALARM_STATE_ACTIVE  ; OP.ALARM.STATE.ACTIVE(FAULTED)
AND MC_LONG_AXIS_ERR  ; LONG.AXIS.ERROR.EXISTS
AND MC_LONG_AXIS_DRV_OL  ; MC.LONG.AXIS.DRIVE.OVERLOAD.FAULT
OUT W115.02
; rung 73
LD OP_ALARM_STATE_ACTIVE  ; OP.ALARM.STATE.ACTIVE(FAULTED)
AND MC_LONG_AXIS_ERR  ; LONG.AXIS.ERROR.EXISTS
AND MC_LONG_AXIS_TEMP_FLT  ; MC.LONG.AXIS.DRIVE.OVER.TEMPERATURE.FAULT
OUT W115.03
; rung 74
LD OP_ALARM_STATE_ACTIVE  ; OP.ALARM.STATE.ACTIVE(FAULTED)
AND MC_LONG_AXIS_ERR  ; LONG.AXIS.ERROR.EXISTS
AND MC_LONG_AXIS_DRV_WRN  ; MC.LONG.AXIS.DRIVE.WARNING.[FAULT EXISTS]
OUT W115.04

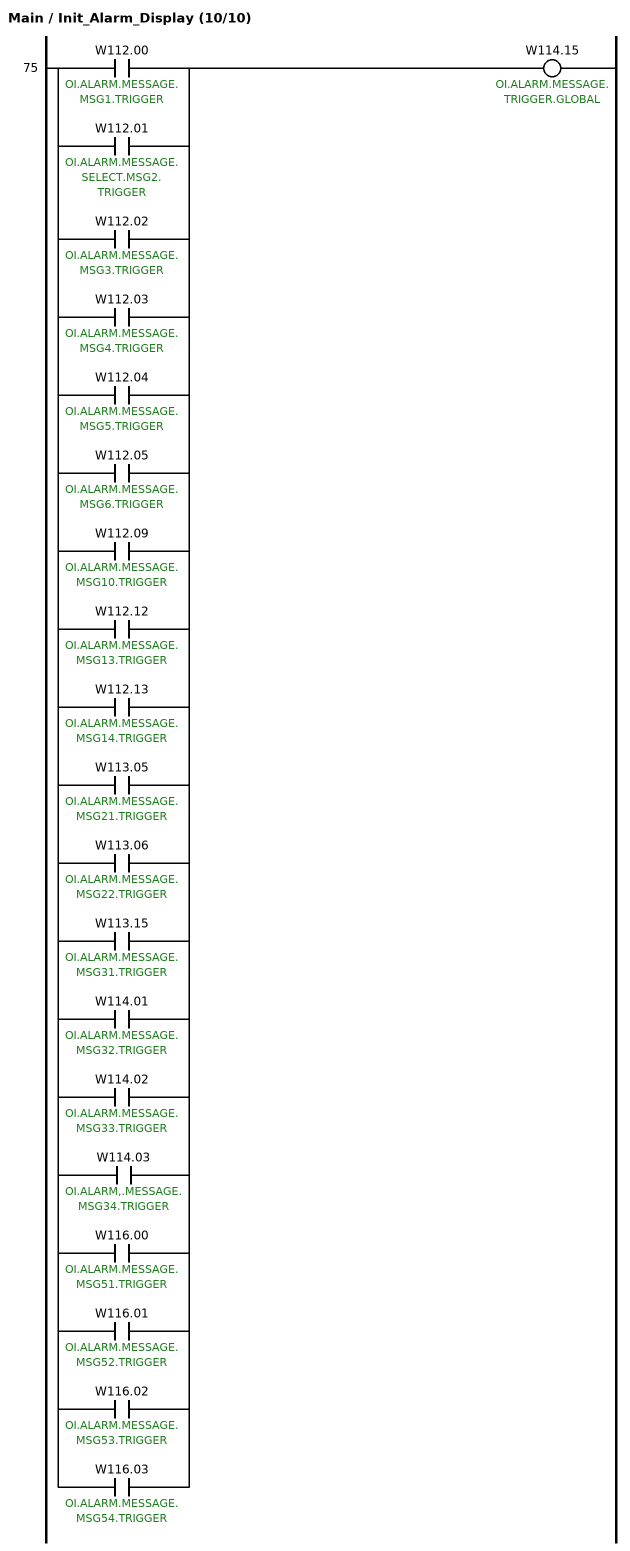
; rung 75
LD W112.00  ; OI.ALARM.MESSAGE.MSG1.TRIGGER
OR W112.01  ; OI.ALARM.MESSAGE.SELECT.MSG2.TRIGGER
OR W112.02  ; OI.ALARM.MESSAGE.MSG3.TRIGGER
OR W112.03  ; OI.ALARM.MESSAGE.MSG4.TRIGGER
OR W112.04  ; OI.ALARM.MESSAGE.MSG5.TRIGGER
OR W112.05  ; OI.ALARM.MESSAGE.MSG6.TRIGGER
OR W112.09  ; OI.ALARM.MESSAGE.MSG10.TRIGGER
OR W112.12  ; OI.ALARM.MESSAGE.MSG13.TRIGGER
OR W112.13  ; OI.ALARM.MESSAGE.MSG14.TRIGGER
OR W113.05  ; OI.ALARM.MESSAGE.MSG21.TRIGGER
OR W113.06  ; OI.ALARM.MESSAGE.MSG22.TRIGGER
OR W113.15  ; OI.ALARM.MESSAGE.MSG31.TRIGGER
OR W114.01  ; OI.ALARM.MESSAGE.MSG32.TRIGGER
OR W114.02  ; OI.ALARM.MESSAGE.MSG33.TRIGGER
OR W114.03  ; OI.ALARM,.MESSAGE.MSG34.TRIGGER
OR W116.00  ; OI.ALARM.MESSAGE.MSG51.TRIGGER
OR W116.01  ; OI.ALARM.MESSAGE.MSG52.TRIGGER
OR W116.02  ; OI.ALARM.MESSAGE.MSG53.TRIGGER
OR W116.03  ; OI.ALARM.MESSAGE.MSG54.TRIGGER
OUT W114.15  ; OI.ALARM.MESSAGE.TRIGGER.GLOBAL

### Section Pgm_Chk

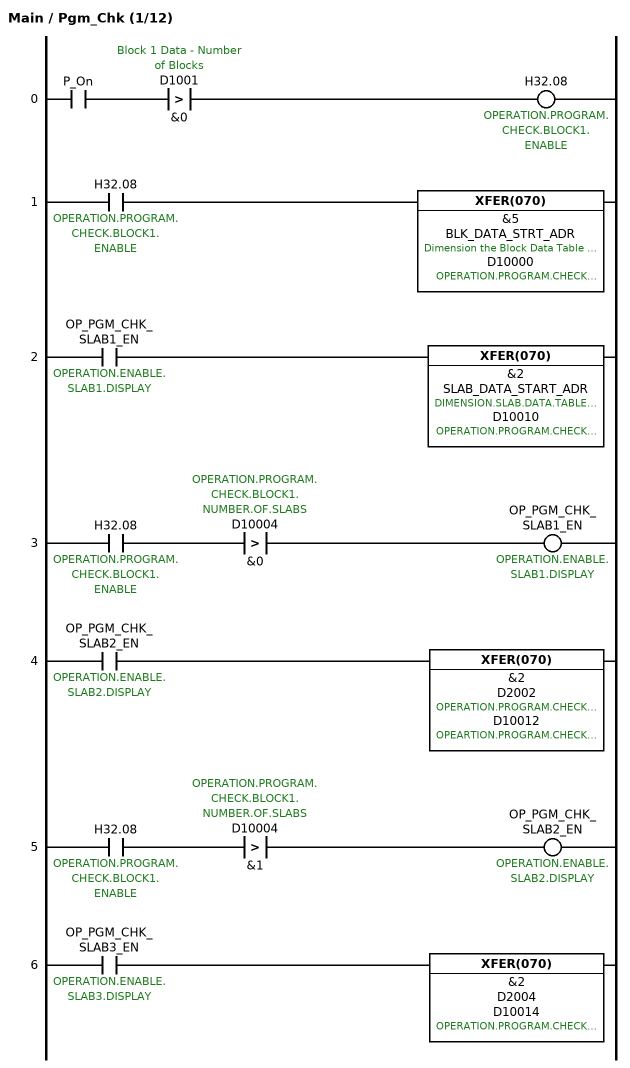
; rung 0
LD P_On
AND>(320) D1001 &0  ; Block 1 Data - Number of Blocks
OUT H32.08  ; OPERATION.PROGRAM.CHECK.BLOCK1.ENABLE
; rung 1
LD H32.08  ; OPERATION.PROGRAM.CHECK.BLOCK1.ENABLE
XFER(070) &5 BLK_DATA_STRT_ADR D10000  ; Dimension the Block Data Table - Start Address, OPERATION.PROGRAM.CHECK.BLOCK1.BLOCK.HEIGHT
; rung 2
LD OP_PGM_CHK_SLAB1_EN  ; OPERATION.ENABLE.SLAB1.DISPLAY
XFER(070) &2 SLAB_DATA_START_ADR D10010  ; DIMENSION.SLAB.DATA.TABLE.START.ADDRESS, OPERATION.PROGRAM.CHECK.BLOCK1.SLAB1.SIZE
; rung 3
LD H32.08  ; OPERATION.PROGRAM.CHECK.BLOCK1.ENABLE
AND>(320) D10004 &0  ; OPERATION.PROGRAM.CHECK.BLOCK1.NUMBER.OF.SLABS
OUT OP_PGM_CHK_SLAB1_EN  ; OPERATION.ENABLE.SLAB1.DISPLAY
; rung 4
LD OP_PGM_CHK_SLAB2_EN  ; OPERATION.ENABLE.SLAB2.DISPLAY
XFER(070) &2 D2002 D10012  ; OPERATION.PROGRAM.CHECK.BLOCK1.SLAB2.SIZE, OPEARTION.PROGRAM.CHECK.BLOCK1SLAB2.SIZE
; rung 5
LD H32.08  ; OPERATION.PROGRAM.CHECK.BLOCK1.ENABLE
AND>(320) D10004 &1  ; OPERATION.PROGRAM.CHECK.BLOCK1.NUMBER.OF.SLABS
OUT OP_PGM_CHK_SLAB2_EN  ; OPERATION.ENABLE.SLAB2.DISPLAY
; rung 6
LD OP_PGM_CHK_SLAB3_EN  ; OPERATION.ENABLE.SLAB3.DISPLAY
XFER(070) &2 D2004 D10014  ; OPERATION.PROGRAM.CHECK.BLOCK1.SLAB3.SIZE

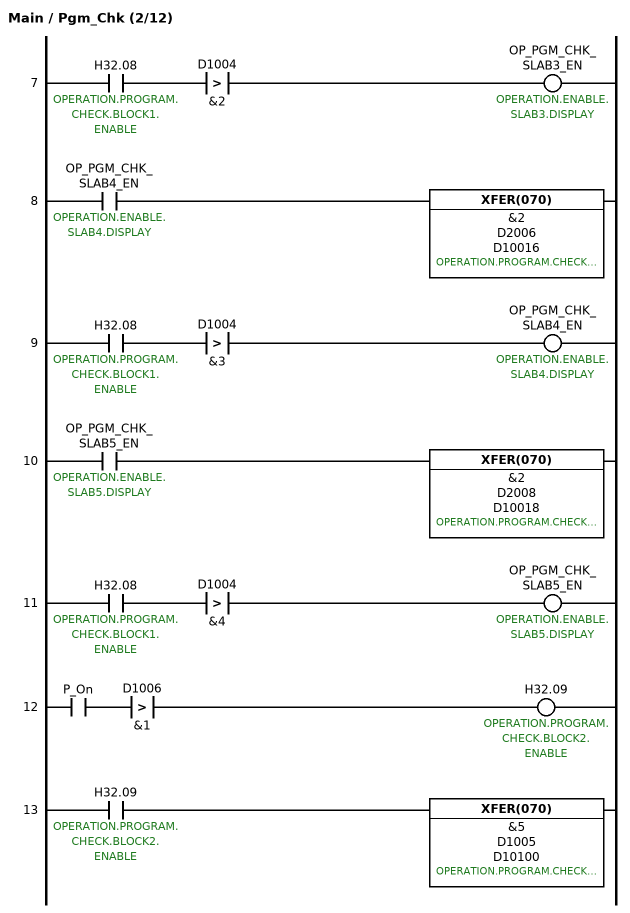
; rung 7
LD H32.08  ; OPERATION.PROGRAM.CHECK.BLOCK1.ENABLE
AND>(320) D1004 &2
OUT OP_PGM_CHK_SLAB3_EN  ; OPERATION.ENABLE.SLAB3.DISPLAY
; rung 8
LD OP_PGM_CHK_SLAB4_EN  ; OPERATION.ENABLE.SLAB4.DISPLAY
XFER(070) &2 D2006 D10016  ; OPERATION.PROGRAM.CHECK.BLOCK1.SLAB4.SIZE
; rung 9
LD H32.08  ; OPERATION.PROGRAM.CHECK.BLOCK1.ENABLE
AND>(320) D1004 &3
OUT OP_PGM_CHK_SLAB4_EN  ; OPERATION.ENABLE.SLAB4.DISPLAY
; rung 10
LD OP_PGM_CHK_SLAB5_EN  ; OPERATION.ENABLE.SLAB5.DISPLAY
XFER(070) &2 D2008 D10018  ; OPERATION.PROGRAM.CHECK.BLOCK1.SLAB5.SIZE
; rung 11
LD H32.08  ; OPERATION.PROGRAM.CHECK.BLOCK1.ENABLE
AND>(320) D1004 &4
OUT OP_PGM_CHK_SLAB5_EN  ; OPERATION.ENABLE.SLAB5.DISPLAY
; rung 12
LD P_On
AND>(320) D1006 &1
OUT H32.09  ; OPERATION.PROGRAM.CHECK.BLOCK2.ENABLE
; rung 13
LD H32.09  ; OPERATION.PROGRAM.CHECK.BLOCK2.ENABLE
XFER(070) &5 D1005 D10100  ; OPERATION.PROGRAM.CHECK.BLOCK2.BLOCK.HEIGHT

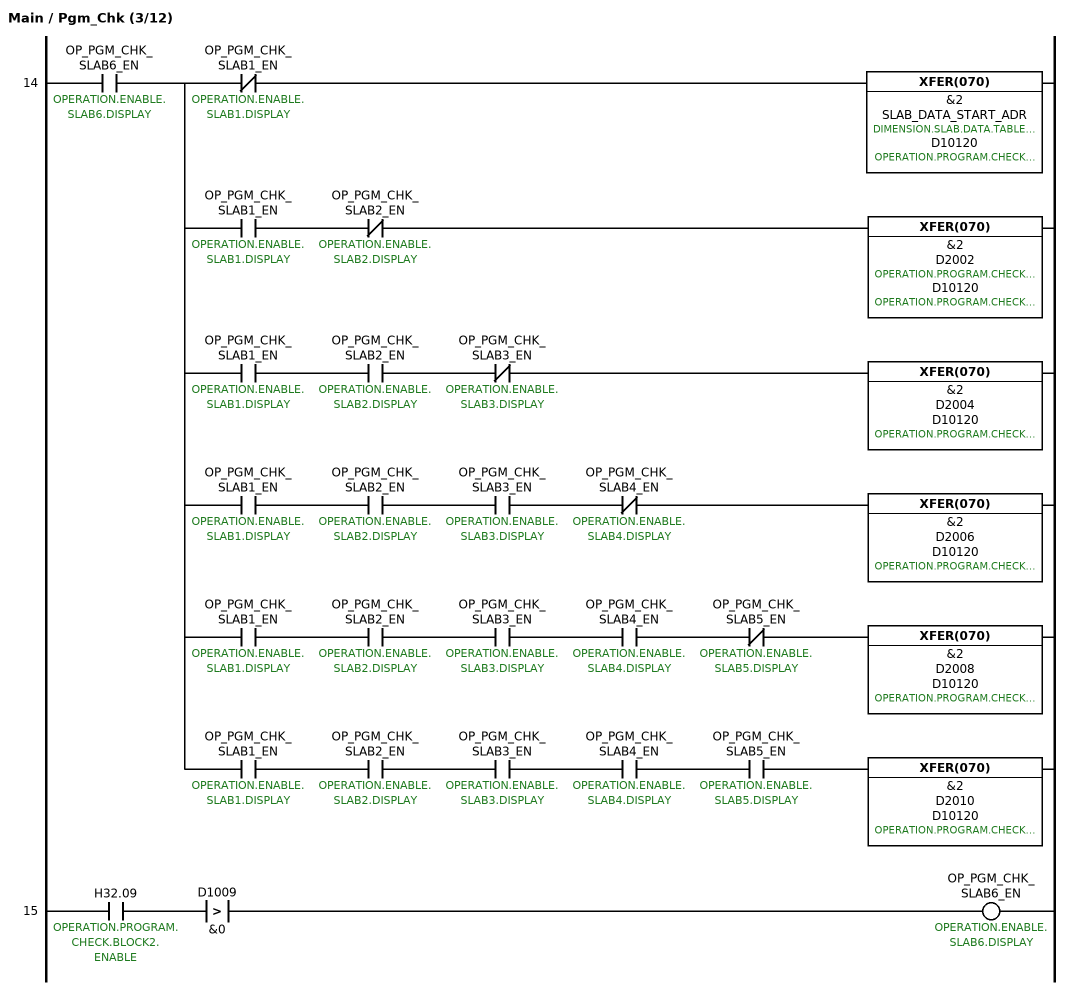
; rung 14
LD OP_PGM_CHK_SLAB6_EN  ; OPERATION.ENABLE.SLAB6.DISPLAY
OUT TR0
ANDNOT OP_PGM_CHK_SLAB1_EN  ; OPERATION.ENABLE.SLAB1.DISPLAY
XFER(070) &2 SLAB_DATA_START_ADR D10120  ; DIMENSION.SLAB.DATA.TABLE.START.ADDRESS, OPERATION.PROGRAM.CHECK.BLOCK2.SLAB1.SIZE
LD TR0
AND OP_PGM_CHK_SLAB1_EN  ; OPERATION.ENABLE.SLAB1.DISPLAY
ANDNOT OP_PGM_CHK_SLAB2_EN  ; OPERATION.ENABLE.SLAB2.DISPLAY
XFER(070) &2 D2002 D10120  ; OPERATION.PROGRAM.CHECK.BLOCK1.SLAB2.SIZE, OPERATION.PROGRAM.CHECK.BLOCK2.SLAB1.SIZE
LD TR0
AND OP_PGM_CHK_SLAB1_EN  ; OPERATION.ENABLE.SLAB1.DISPLAY
AND OP_PGM_CHK_SLAB2_EN  ; OPERATION.ENABLE.SLAB2.DISPLAY
ANDNOT OP_PGM_CHK_SLAB3_EN  ; OPERATION.ENABLE.SLAB3.DISPLAY
XFER(070) &2 D2004 D10120  ; OPERATION.PROGRAM.CHECK.BLOCK2.SLAB1.SIZE
LD TR0
AND OP_PGM_CHK_SLAB1_EN  ; OPERATION.ENABLE.SLAB1.DISPLAY
AND OP_PGM_CHK_SLAB2_EN  ; OPERATION.ENABLE.SLAB2.DISPLAY
AND OP_PGM_CHK_SLAB3_EN  ; OPERATION.ENABLE.SLAB3.DISPLAY
ANDNOT OP_PGM_CHK_SLAB4_EN  ; OPERATION.ENABLE.SLAB4.DISPLAY
XFER(070) &2 D2006 D10120  ; OPERATION.PROGRAM.CHECK.BLOCK2.SLAB1.SIZE
LD TR0
AND OP_PGM_CHK_SLAB1_EN  ; OPERATION.ENABLE.SLAB1.DISPLAY
AND OP_PGM_CHK_SLAB2_EN  ; OPERATION.ENABLE.SLAB2.DISPLAY
AND OP_PGM_CHK_SLAB3_EN  ; OPERATION.ENABLE.SLAB3.DISPLAY
AND OP_PGM_CHK_SLAB4_EN  ; OPERATION.ENABLE.SLAB4.DISPLAY
ANDNOT OP_PGM_CHK_SLAB5_EN  ; OPERATION.ENABLE.SLAB5.DISPLAY
XFER(070) &2 D2008 D10120  ; OPERATION.PROGRAM.CHECK.BLOCK2.SLAB1.SIZE
LD TR0
AND OP_PGM_CHK_SLAB1_EN  ; OPERATION.ENABLE.SLAB1.DISPLAY
AND OP_PGM_CHK_SLAB2_EN  ; OPERATION.ENABLE.SLAB2.DISPLAY
AND OP_PGM_CHK_SLAB3_EN  ; OPERATION.ENABLE.SLAB3.DISPLAY
AND OP_PGM_CHK_SLAB4_EN  ; OPERATION.ENABLE.SLAB4.DISPLAY
AND OP_PGM_CHK_SLAB5_EN  ; OPERATION.ENABLE.SLAB5.DISPLAY
XFER(070) &2 D2010 D10120  ; OPERATION.PROGRAM.CHECK.BLOCK2.SLAB1.SIZE
; rung 15
LD H32.09  ; OPERATION.PROGRAM.CHECK.BLOCK2.ENABLE
AND>(320) D1009 &0
OUT OP_PGM_CHK_SLAB6_EN  ; OPERATION.ENABLE.SLAB6.DISPLAY

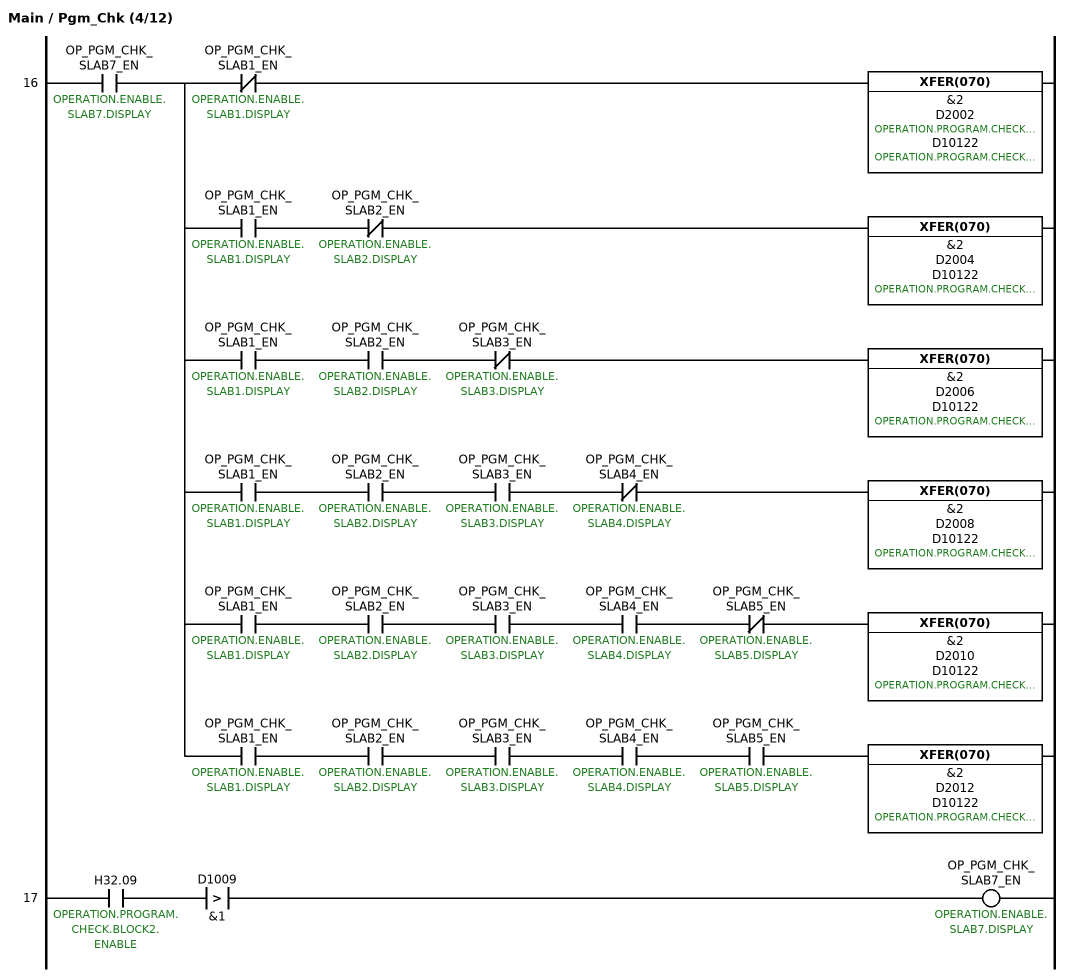
; rung 16
LD OP_PGM_CHK_SLAB7_EN  ; OPERATION.ENABLE.SLAB7.DISPLAY
OUT TR0
ANDNOT OP_PGM_CHK_SLAB1_EN  ; OPERATION.ENABLE.SLAB1.DISPLAY
XFER(070) &2 D2002 D10122  ; OPERATION.PROGRAM.CHECK.BLOCK1.SLAB2.SIZE, OPERATION.PROGRAM.CHECK.BLOCK2.SLAB2.SIZE
LD TR0
AND OP_PGM_CHK_SLAB1_EN  ; OPERATION.ENABLE.SLAB1.DISPLAY
ANDNOT OP_PGM_CHK_SLAB2_EN  ; OPERATION.ENABLE.SLAB2.DISPLAY
XFER(070) &2 D2004 D10122  ; OPERATION.PROGRAM.CHECK.BLOCK2.SLAB2.SIZE
LD TR0
AND OP_PGM_CHK_SLAB1_EN  ; OPERATION.ENABLE.SLAB1.DISPLAY
AND OP_PGM_CHK_SLAB2_EN  ; OPERATION.ENABLE.SLAB2.DISPLAY
ANDNOT OP_PGM_CHK_SLAB3_EN  ; OPERATION.ENABLE.SLAB3.DISPLAY
XFER(070) &2 D2006 D10122  ; OPERATION.PROGRAM.CHECK.BLOCK2.SLAB2.SIZE
LD TR0
AND OP_PGM_CHK_SLAB1_EN  ; OPERATION.ENABLE.SLAB1.DISPLAY
AND OP_PGM_CHK_SLAB2_EN  ; OPERATION.ENABLE.SLAB2.DISPLAY
AND OP_PGM_CHK_SLAB3_EN  ; OPERATION.ENABLE.SLAB3.DISPLAY
ANDNOT OP_PGM_CHK_SLAB4_EN  ; OPERATION.ENABLE.SLAB4.DISPLAY
XFER(070) &2 D2008 D10122  ; OPERATION.PROGRAM.CHECK.BLOCK2.SLAB2.SIZE
LD TR0
AND OP_PGM_CHK_SLAB1_EN  ; OPERATION.ENABLE.SLAB1.DISPLAY
AND OP_PGM_CHK_SLAB2_EN  ; OPERATION.ENABLE.SLAB2.DISPLAY
AND OP_PGM_CHK_SLAB3_EN  ; OPERATION.ENABLE.SLAB3.DISPLAY
AND OP_PGM_CHK_SLAB4_EN  ; OPERATION.ENABLE.SLAB4.DISPLAY
ANDNOT OP_PGM_CHK_SLAB5_EN  ; OPERATION.ENABLE.SLAB5.DISPLAY
XFER(070) &2 D2010 D10122  ; OPERATION.PROGRAM.CHECK.BLOCK2.SLAB2.SIZE
LD TR0
AND OP_PGM_CHK_SLAB1_EN  ; OPERATION.ENABLE.SLAB1.DISPLAY
AND OP_PGM_CHK_SLAB2_EN  ; OPERATION.ENABLE.SLAB2.DISPLAY
AND OP_PGM_CHK_SLAB3_EN  ; OPERATION.ENABLE.SLAB3.DISPLAY
AND OP_PGM_CHK_SLAB4_EN  ; OPERATION.ENABLE.SLAB4.DISPLAY
AND OP_PGM_CHK_SLAB5_EN  ; OPERATION.ENABLE.SLAB5.DISPLAY
XFER(070) &2 D2012 D10122  ; OPERATION.PROGRAM.CHECK.BLOCK2.SLAB2.SIZE
; rung 17
LD H32.09  ; OPERATION.PROGRAM.CHECK.BLOCK2.ENABLE
AND>(320) D1009 &1
OUT OP_PGM_CHK_SLAB7_EN  ; OPERATION.ENABLE.SLAB7.DISPLAY

